(* IEC 61131-3 sources: eCockpitGit/test_project/src/%PLC%PFC100_2ETH_ECO/%PLOG%Plc Logic/%APP%Application, 3 files *)

(* ---- %POU%ProjectBeforeBoot.st ---- *)
PROGRAM ProjectBeforeBoot
VAR
END_VAR

(*%!%__DELIMITER__%!%*)
GMemory.dynamicSize			:=		3000000;
W8100();

(* ---- %POU%ProjectDuringBoot.st ---- *)
PROGRAM ProjectDuringBoot
VAR
END_VAR
VAR_IN_OUT
	pouSpeed		:WORD;
END_VAR

(*%!%__DELIMITER__%!%*)
//GMod.modMan.registerModule(parentModule:=ADR(GMod.modMan),moduleBuffer:=ADR(W8100.pms),access:=GUsers.userAndPublicRead,subID:=0,mid:=0,client:=0);

(* ---- %POU%W8100.st ---- *)
PROGRAM W8100
VAR
	boot			:BOOL;
END_VAR

// VAR_OUTPUT
// 	pms				:FB_PMS := (_name:=ADR('PMS System'));
// END_VAR
(*%!%__DELIMITER__%!%*)
boot				:=		PRG_BootManager.bootFinished;
